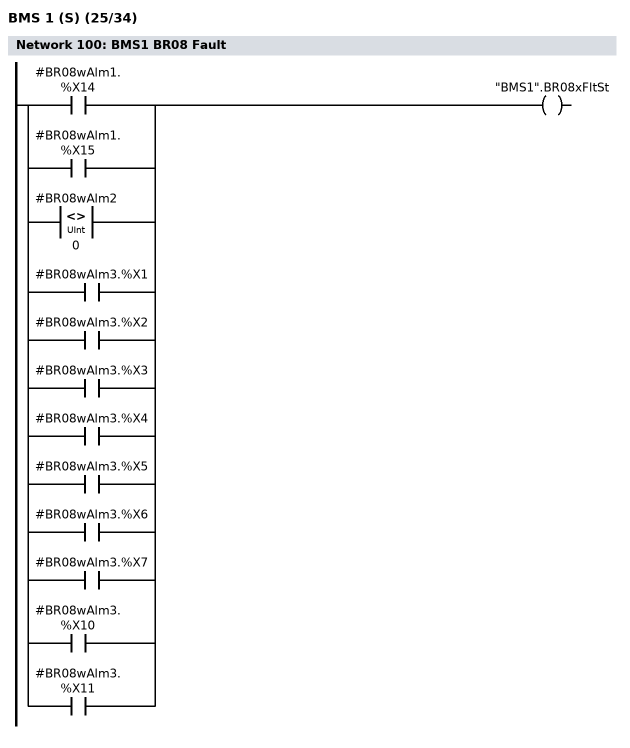
   RUNG wire#powerrail
      Contact( #BR08wAlm1.%X14 )
      wire#w1
      Coil( "BMS1".BR08xFltSt )
   END_RUNG
   RUNG wire#powerrail
      Contact( #BR08wAlm1.%X15 )
   END_RUNG wire#w1
   RUNG wire#powerrail
      { S7_Templates := "SrcType := UInt" } NE_Contact(in1 := #BR08wAlm2, in2 := 0)
   END_RUNG wire#w1
   RUNG wire#powerrail
      Contact( #BR08wAlm3.%X1 )
   END_RUNG wire#w1
   RUNG wire#powerrail
      Contact( #BR08wAlm3.%X2 )
   END_RUNG wire#w1
   RUNG wire#powerrail
      Contact( #BR08wAlm3.%X3 )
   END_RUNG wire#w1
   RUNG wire#powerrail
      Contact( #BR08wAlm3.%X4 )
   END_RUNG wire#w1
   RUNG wire#powerrail
      Contact( #BR08wAlm3.%X5 )
   END_RUNG wire#w1
   RUNG wire#powerrail
      Contact( #BR08wAlm3.%X6 )
   END_RUNG wire#w1
   RUNG wire#powerrail
      Contact( #BR08wAlm3.%X7 )
   END_RUNG wire#w1
   RUNG wire#powerrail
      Contact( #BR08wAlm3.%X10 )
   END_RUNG wire#w1
   RUNG wire#powerrail
      Contact( #BR08wAlm3.%X11 )
   END_RUNG wire#w1
   // the same network as SCL:
   "BMS1".BR08xFltSt := #BR08wAlm1.%X14 OR #BR08wAlm1.%X15 OR (#BR08wAlm2 <> 0) OR #BR08wAlm3.%X1 OR #BR08wAlm3.%X2 OR #BR08wAlm3.%X3 OR #BR08wAlm3.%X4 OR #BR08wAlm3.%X5 OR #BR08wAlm3.%X6 OR #BR08wAlm3.%X7 OR #BR08wAlm3.%X10 OR #BR08wAlm3.%X11;
END_REGION

REGION Network 101: BMS1 BR08 Alarm
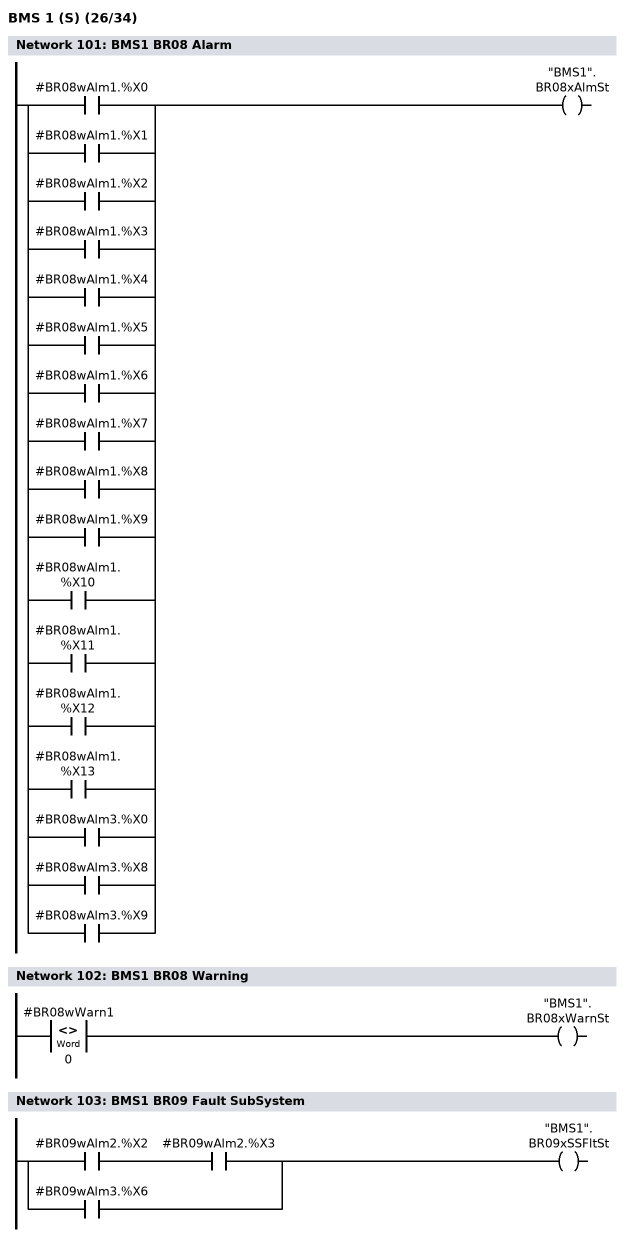
   RUNG wire#powerrail
      Contact( #BR08wAlm1.%X0 )
      wire#w1
      Coil( "BMS1".BR08xAlmSt )
   END_RUNG
   RUNG wire#powerrail
      Contact( #BR08wAlm1.%X1 )
   END_RUNG wire#w1
   RUNG wire#powerrail
      Contact( #BR08wAlm1.%X2 )
   END_RUNG wire#w1
   RUNG wire#powerrail
      Contact( #BR08wAlm1.%X3 )
   END_RUNG wire#w1
   RUNG wire#powerrail
      Contact( #BR08wAlm1.%X4 )
   END_RUNG wire#w1
   RUNG wire#powerrail
      Contact( #BR08wAlm1.%X5 )
   END_RUNG wire#w1
   RUNG wire#powerrail
      Contact( #BR08wAlm1.%X6 )
   END_RUNG wire#w1
   RUNG wire#powerrail
      Contact( #BR08wAlm1.%X7 )
   END_RUNG wire#w1
   RUNG wire#powerrail
      Contact( #BR08wAlm1.%X8 )
   END_RUNG wire#w1
   RUNG wire#powerrail
      Contact( #BR08wAlm1.%X9 )
   END_RUNG wire#w1
   RUNG wire#powerrail
      Contact( #BR08wAlm1.%X10 )
   END_RUNG wire#w1
   RUNG wire#powerrail
      Contact( #BR08wAlm1.%X11 )
   END_RUNG wire#w1
   RUNG wire#powerrail
      Contact( #BR08wAlm1.%X12 )
   END_RUNG wire#w1
   RUNG wire#powerrail
      Contact( #BR08wAlm1.%X13 )
   END_RUNG wire#w1
   RUNG wire#powerrail
      Contact( #BR08wAlm3.%X0 )
   END_RUNG wire#w1
   RUNG wire#powerrail
      Contact( #BR08wAlm3.%X8 )
   END_RUNG wire#w1
   RUNG wire#powerrail
      Contact( #BR08wAlm3.%X9 )
   END_RUNG wire#w1
   // the same network as SCL:
   "BMS1".BR08xAlmSt := #BR08wAlm1.%X0 OR #BR08wAlm1.%X1 OR #BR08wAlm1.%X2 OR #BR08wAlm1.%X3 OR #BR08wAlm1.%X4 OR #BR08wAlm1.%X5 OR #BR08wAlm1.%X6 OR #BR08wAlm1.%X7 OR #BR08wAlm1.%X8 OR #BR08wAlm1.%X9 OR #BR08wAlm1.%X10 OR #BR08wAlm1.%X11 OR #BR08wAlm1.%X12 OR #BR08wAlm1.%X13 OR #BR08wAlm3.%X0 OR #BR08wAlm3.%X8 OR #BR08wAlm3.%X9;
END_REGION

REGION Network 102: BMS1 BR08 Warning
   RUNG wire#powerrail
      { S7_Templates := "SrcType := Word" } NE_Contact(in1 := #BR08wWarn1, in2 := 0)
      Coil( "BMS1".BR08xWarnSt )
   END_RUNG
   // the same network as SCL:
   "BMS1".BR08xWarnSt := #BR08wWarn1 <> 0;
END_REGION

REGION Network 103: BMS1 BR09 Fault SubSystem
   RUNG wire#powerrail
      Contact( #BR09wAlm2.%X2 )
      Contact( #BR09wAlm2.%X3 )
      wire#w1
      Coil( "BMS1".BR09xSSFltSt )
   END_RUNG
   RUNG wire#powerrail
      Contact( #BR09wAlm3.%X6 )
   END_RUNG wire#w1
   // the same network as SCL:
   "BMS1".BR09xSSFltSt := (#BR09wAlm2.%X2 AND #BR09wAlm2.%X3) OR #BR09wAlm3.%X6;
END_REGION

REGION Network 104: BMS1 BR09 Fault
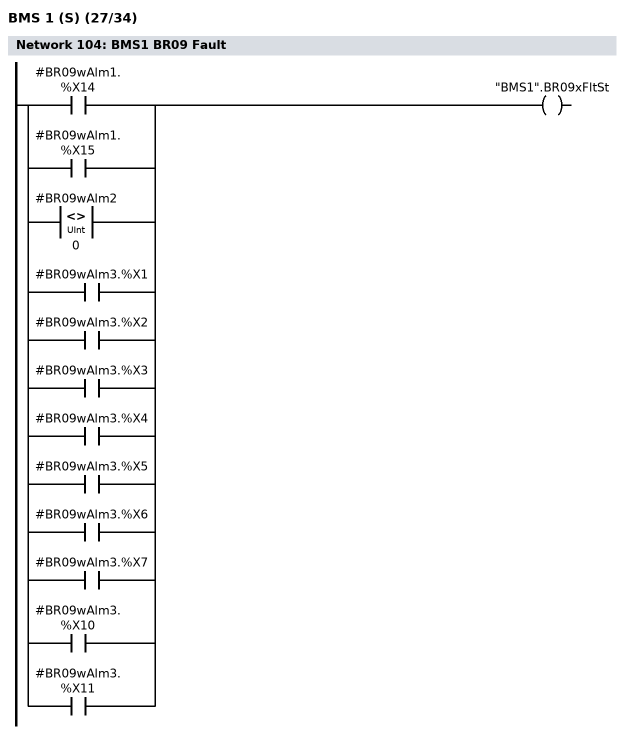
   RUNG wire#powerrail
      Contact( #BR09wAlm1.%X14 )
      wire#w1
      Coil( "BMS1".BR09xFltSt )
   END_RUNG
   RUNG wire#powerrail
      Contact( #BR09wAlm1.%X15 )
   END_RUNG wire#w1
   RUNG wire#powerrail
      { S7_Templates := "SrcType := UInt" } NE_Contact(in1 := #BR09wAlm2, in2 := 0)
   END_RUNG wire#w1
   RUNG wire#powerrail
      Contact( #BR09wAlm3.%X1 )
   END_RUNG wire#w1
   RUNG wire#powerrail
      Contact( #BR09wAlm3.%X2 )
   END_RUNG wire#w1
   RUNG wire#powerrail
      Contact( #BR09wAlm3.%X3 )
   END_RUNG wire#w1
   RUNG wire#powerrail
      Contact( #BR09wAlm3.%X4 )
   END_RUNG wire#w1
   RUNG wire#powerrail
      Contact( #BR09wAlm3.%X5 )
   END_RUNG wire#w1
   RUNG wire#powerrail
      Contact( #BR09wAlm3.%X6 )
   END_RUNG wire#w1
   RUNG wire#powerrail
      Contact( #BR09wAlm3.%X7 )
   END_RUNG wire#w1
   RUNG wire#powerrail
      Contact( #BR09wAlm3.%X10 )
   END_RUNG wire#w1
   RUNG wire#powerrail
      Contact( #BR09wAlm3.%X11 )
   END_RUNG wire#w1
   // the same network as SCL:
   "BMS1".BR09xFltSt := #BR09wAlm1.%X14 OR #BR09wAlm1.%X15 OR (#BR09wAlm2 <> 0) OR #BR09wAlm3.%X1 OR #BR09wAlm3.%X2 OR #BR09wAlm3.%X3 OR #BR09wAlm3.%X4 OR #BR09wAlm3.%X5 OR #BR09wAlm3.%X6 OR #BR09wAlm3.%X7 OR #BR09wAlm3.%X10 OR #BR09wAlm3.%X11;
END_REGION

REGION Network 105: BMS1 BR09 Alarm
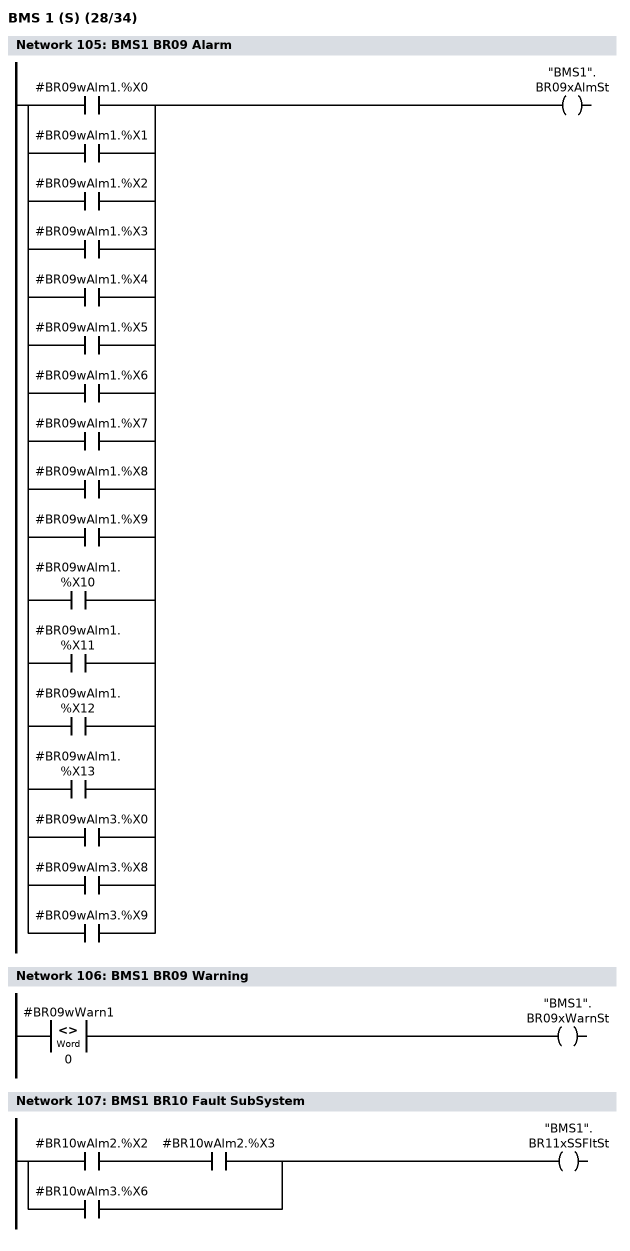
   RUNG wire#powerrail
      Contact( #BR09wAlm1.%X0 )
      wire#w1
      Coil( "BMS1".BR09xAlmSt )
   END_RUNG
   RUNG wire#powerrail
      Contact( #BR09wAlm1.%X1 )
   END_RUNG wire#w1
   RUNG wire#powerrail
      Contact( #BR09wAlm1.%X2 )
   END_RUNG wire#w1
   RUNG wire#powerrail
      Contact( #BR09wAlm1.%X3 )
   END_RUNG wire#w1
   RUNG wire#powerrail
      Contact( #BR09wAlm1.%X4 )
   END_RUNG wire#w1
   RUNG wire#powerrail
      Contact( #BR09wAlm1.%X5 )
   END_RUNG wire#w1
   RUNG wire#powerrail
      Contact( #BR09wAlm1.%X6 )
   END_RUNG wire#w1
   RUNG wire#powerrail
      Contact( #BR09wAlm1.%X7 )
   END_RUNG wire#w1
   RUNG wire#powerrail
      Contact( #BR09wAlm1.%X8 )
   END_RUNG wire#w1
   RUNG wire#powerrail
      Contact( #BR09wAlm1.%X9 )
   END_RUNG wire#w1
   RUNG wire#powerrail
      Contact( #BR09wAlm1.%X10 )
   END_RUNG wire#w1
   RUNG wire#powerrail
      Contact( #BR09wAlm1.%X11 )
   END_RUNG wire#w1
   RUNG wire#powerrail
      Contact( #BR09wAlm1.%X12 )
   END_RUNG wire#w1
   RUNG wire#powerrail
      Contact( #BR09wAlm1.%X13 )
   END_RUNG wire#w1
   RUNG wire#powerrail
      Contact( #BR09wAlm3.%X0 )
   END_RUNG wire#w1
   RUNG wire#powerrail
      Contact( #BR09wAlm3.%X8 )
   END_RUNG wire#w1
   RUNG wire#powerrail
      Contact( #BR09wAlm3.%X9 )
   END_RUNG wire#w1
   // the same network as SCL:
   "BMS1".BR09xAlmSt := #BR09wAlm1.%X0 OR #BR09wAlm1.%X1 OR #BR09wAlm1.%X2 OR #BR09wAlm1.%X3 OR #BR09wAlm1.%X4 OR #BR09wAlm1.%X5 OR #BR09wAlm1.%X6 OR #BR09wAlm1.%X7 OR #BR09wAlm1.%X8 OR #BR09wAlm1.%X9 OR #BR09wAlm1.%X10 OR #BR09wAlm1.%X11 OR #BR09wAlm1.%X12 OR #BR09wAlm1.%X13 OR #BR09wAlm3.%X0 OR #BR09wAlm3.%X8 OR #BR09wAlm3.%X9;
END_REGION

REGION Network 106: BMS1 BR09 Warning
   RUNG wire#powerrail
      { S7_Templates := "SrcType := Word" } NE_Contact(in1 := #BR09wWarn1, in2 := 0)
      Coil( "BMS1".BR09xWarnSt )
   END_RUNG
   // the same network as SCL:
   "BMS1".BR09xWarnSt := #BR09wWarn1 <> 0;
END_REGION

REGION Network 107: BMS1 BR10 Fault SubSystem
   RUNG wire#powerrail
      Contact( #BR10wAlm2.%X2 )
      Contact( #BR10wAlm2.%X3 )
      wire#w1
      Coil( "BMS1".BR11xSSFltSt )
   END_RUNG
   RUNG wire#powerrail
      Contact( #BR10wAlm3.%X6 )
   END_RUNG wire#w1
   // the same network as SCL:
   "BMS1".BR11xSSFltSt := (#BR10wAlm2.%X2 AND #BR10wAlm2.%X3) OR #BR10wAlm3.%X6;
END_REGION

REGION Network 108: BMS1 BR10 Fault
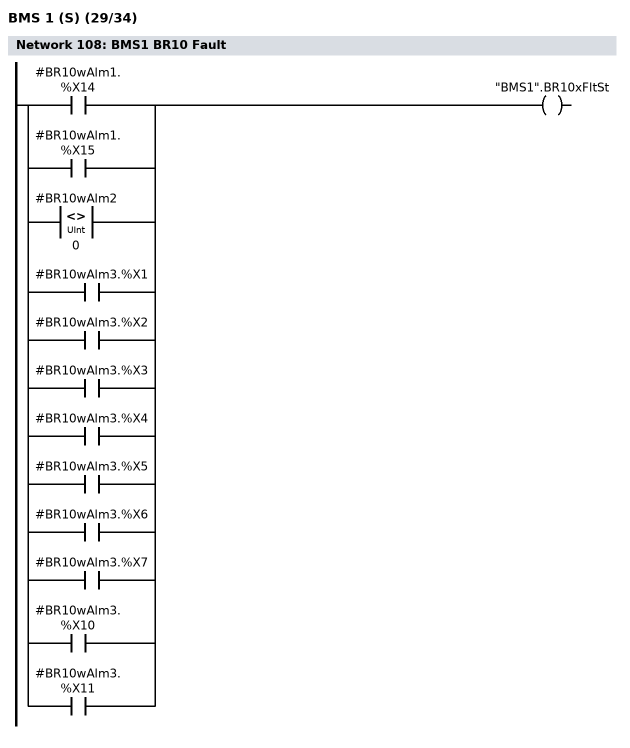
   RUNG wire#powerrail
      Contact( #BR10wAlm1.%X14 )
      wire#w1
      Coil( "BMS1".BR10xFltSt )
   END_RUNG
   RUNG wire#powerrail
      Contact( #BR10wAlm1.%X15 )
   END_RUNG wire#w1
   RUNG wire#powerrail
      { S7_Templates := "SrcType := UInt" } NE_Contact(in1 := #BR10wAlm2, in2 := 0)
   END_RUNG wire#w1
   RUNG wire#powerrail
      Contact( #BR10wAlm3.%X1 )
   END_RUNG wire#w1
   RUNG wire#powerrail
      Contact( #BR10wAlm3.%X2 )
   END_RUNG wire#w1
   RUNG wire#powerrail
      Contact( #BR10wAlm3.%X3 )
   END_RUNG wire#w1
   RUNG wire#powerrail
      Contact( #BR10wAlm3.%X4 )
   END_RUNG wire#w1
   RUNG wire#powerrail
      Contact( #BR10wAlm3.%X5 )
   END_RUNG wire#w1
   RUNG wire#powerrail
      Contact( #BR10wAlm3.%X6 )
   END_RUNG wire#w1
   RUNG wire#powerrail
      Contact( #BR10wAlm3.%X7 )
   END_RUNG wire#w1
   RUNG wire#powerrail
      Contact( #BR10wAlm3.%X10 )
   END_RUNG wire#w1
   RUNG wire#powerrail
      Contact( #BR10wAlm3.%X11 )
   END_RUNG wire#w1
   // the same network as SCL:
   "BMS1".BR10xFltSt := #BR10wAlm1.%X14 OR #BR10wAlm1.%X15 OR (#BR10wAlm2 <> 0) OR #BR10wAlm3.%X1 OR #BR10wAlm3.%X2 OR #BR10wAlm3.%X3 OR #BR10wAlm3.%X4 OR #BR10wAlm3.%X5 OR #BR10wAlm3.%X6 OR #BR10wAlm3.%X7 OR #BR10wAlm3.%X10 OR #BR10wAlm3.%X11;
END_REGION

REGION Network 109: BMS1 BR10 Alarm
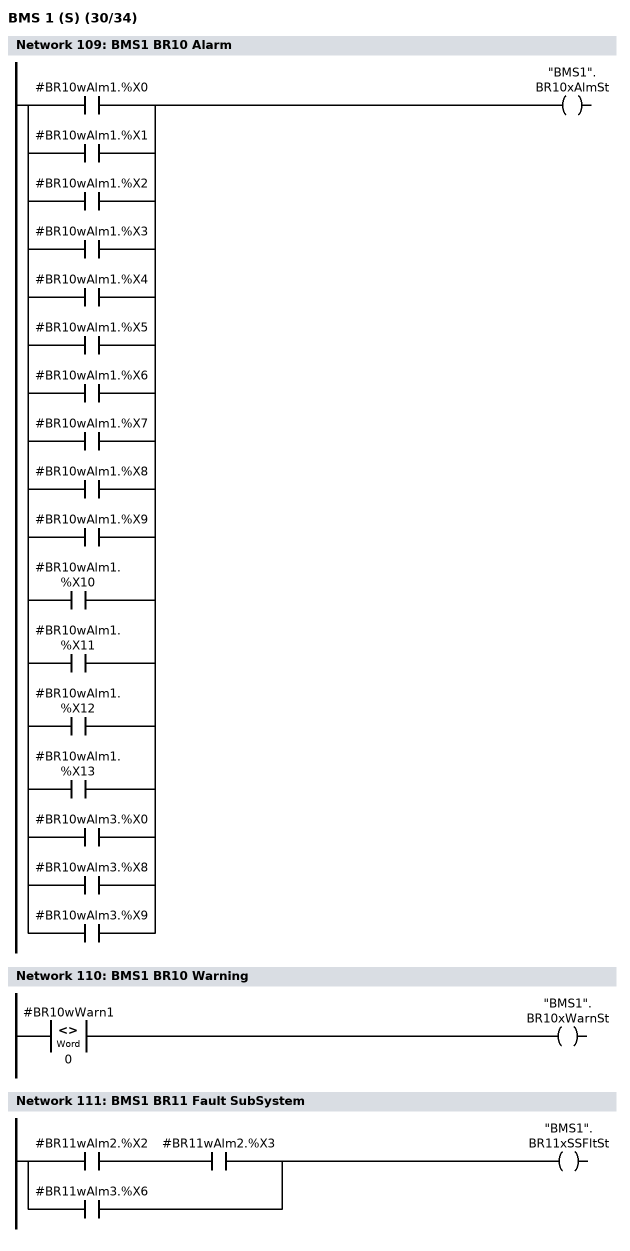
   RUNG wire#powerrail
      Contact( #BR10wAlm1.%X0 )
      wire#w1
      Coil( "BMS1".BR10xAlmSt )
   END_RUNG
   RUNG wire#powerrail
      Contact( #BR10wAlm1.%X1 )
   END_RUNG wire#w1
   RUNG wire#powerrail
      Contact( #BR10wAlm1.%X2 )
   END_RUNG wire#w1
   RUNG wire#powerrail
      Contact( #BR10wAlm1.%X3 )
   END_RUNG wire#w1
   RUNG wire#powerrail
      Contact( #BR10wAlm1.%X4 )
   END_RUNG wire#w1
   RUNG wire#powerrail
      Contact( #BR10wAlm1.%X5 )
   END_RUNG wire#w1
   RUNG wire#powerrail
      Contact( #BR10wAlm1.%X6 )
   END_RUNG wire#w1
   RUNG wire#powerrail
      Contact( #BR10wAlm1.%X7 )
   END_RUNG wire#w1
   RUNG wire#powerrail
      Contact( #BR10wAlm1.%X8 )
   END_RUNG wire#w1
   RUNG wire#powerrail
      Contact( #BR10wAlm1.%X9 )
   END_RUNG wire#w1
   RUNG wire#powerrail
      Contact( #BR10wAlm1.%X10 )
   END_RUNG wire#w1
   RUNG wire#powerrail
      Contact( #BR10wAlm1.%X11 )
   END_RUNG wire#w1
   RUNG wire#powerrail
      Contact( #BR10wAlm1.%X12 )
   END_RUNG wire#w1
   RUNG wire#powerrail
      Contact( #BR10wAlm1.%X13 )
   END_RUNG wire#w1
   RUNG wire#powerrail
      Contact( #BR10wAlm3.%X0 )
   END_RUNG wire#w1
   RUNG wire#powerrail
      Contact( #BR10wAlm3.%X8 )
   END_RUNG wire#w1
   RUNG wire#powerrail
      Contact( #BR10wAlm3.%X9 )
   END_RUNG wire#w1
   // the same network as SCL:
   "BMS1".BR10xAlmSt := #BR10wAlm1.%X0 OR #BR10wAlm1.%X1 OR #BR10wAlm1.%X2 OR #BR10wAlm1.%X3 OR #BR10wAlm1.%X4 OR #BR10wAlm1.%X5 OR #BR10wAlm1.%X6 OR #BR10wAlm1.%X7 OR #BR10wAlm1.%X8 OR #BR10wAlm1.%X9 OR #BR10wAlm1.%X10 OR #BR10wAlm1.%X11 OR #BR10wAlm1.%X12 OR #BR10wAlm1.%X13 OR #BR10wAlm3.%X0 OR #BR10wAlm3.%X8 OR #BR10wAlm3.%X9;
END_REGION

REGION Network 110: BMS1 BR10 Warning
   RUNG wire#powerrail
      { S7_Templates := "SrcType := Word" } NE_Contact(in1 := #BR10wWarn1, in2 := 0)
      Coil( "BMS1".BR10xWarnSt )
   END_RUNG
   // the same network as SCL:
   "BMS1".BR10xWarnSt := #BR10wWarn1 <> 0;
END_REGION

REGION Network 111: BMS1 BR11 Fault SubSystem
   RUNG wire#powerrail
      Contact( #BR11wAlm2.%X2 )
      Contact( #BR11wAlm2.%X3 )
      wire#w1
      Coil( "BMS1".BR11xSSFltSt )
   END_RUNG
   RUNG wire#powerrail
      Contact( #BR11wAlm3.%X6 )
   END_RUNG wire#w1
   // the same network as SCL:
   "BMS1".BR11xSSFltSt := (#BR11wAlm2.%X2 AND #BR11wAlm2.%X3) OR #BR11wAlm3.%X6;
END_REGION

REGION Network 112: BMS1 BR11 Fault
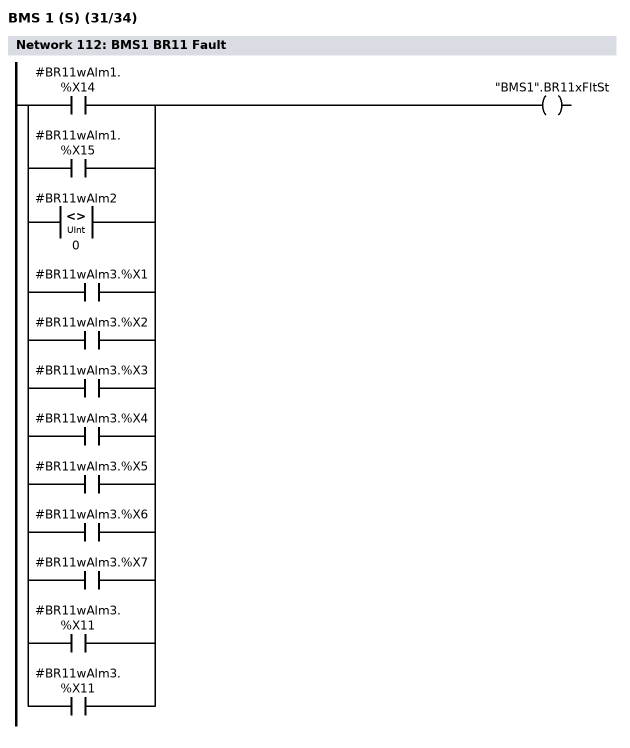
   RUNG wire#powerrail
      Contact( #BR11wAlm1.%X14 )
      wire#w1
      Coil( "BMS1".BR11xFltSt )
   END_RUNG
   RUNG wire#powerrail
      Contact( #BR11wAlm1.%X15 )
   END_RUNG wire#w1
   RUNG wire#powerrail
      { S7_Templates := "SrcType := UInt" } NE_Contact(in1 := #BR11wAlm2, in2 := 0)
   END_RUNG wire#w1
   RUNG wire#powerrail
      Contact( #BR11wAlm3.%X1 )
   END_RUNG wire#w1
   RUNG wire#powerrail
      Contact( #BR11wAlm3.%X2 )
   END_RUNG wire#w1
   RUNG wire#powerrail
      Contact( #BR11wAlm3.%X3 )
   END_RUNG wire#w1
   RUNG wire#powerrail
      Contact( #BR11wAlm3.%X4 )
   END_RUNG wire#w1
   RUNG wire#powerrail
      Contact( #BR11wAlm3.%X5 )
   END_RUNG wire#w1
   RUNG wire#powerrail
      Contact( #BR11wAlm3.%X6 )
   END_RUNG wire#w1
   RUNG wire#powerrail
      Contact( #BR11wAlm3.%X7 )
   END_RUNG wire#w1
   RUNG wire#powerrail
      Contact( #BR11wAlm3.%X11 )
   END_RUNG wire#w1
   RUNG wire#powerrail
      Contact( #BR11wAlm3.%X11 )
   END_RUNG wire#w1
   // the same network as SCL:
   "BMS1".BR11xFltSt := #BR11wAlm1.%X14 OR #BR11wAlm1.%X15 OR (#BR11wAlm2 <> 0) OR #BR11wAlm3.%X1 OR #BR11wAlm3.%X2 OR #BR11wAlm3.%X3 OR #BR11wAlm3.%X4 OR #BR11wAlm3.%X5 OR #BR11wAlm3.%X6 OR #BR11wAlm3.%X7 OR #BR11wAlm3.%X11 OR #BR11wAlm3.%X11;
END_REGION

REGION Network 113: BMS1 BR11 Alarm
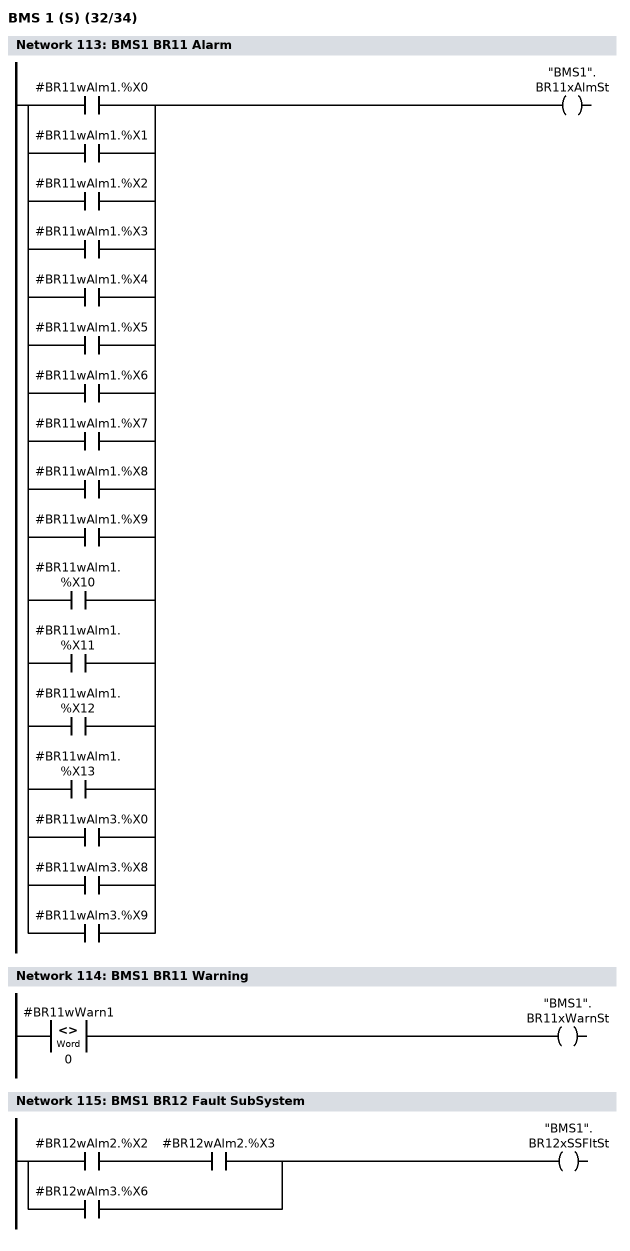
   RUNG wire#powerrail
      Contact( #BR11wAlm1.%X0 )
      wire#w1
      Coil( "BMS1".BR11xAlmSt )
   END_RUNG
   RUNG wire#powerrail
      Contact( #BR11wAlm1.%X1 )
   END_RUNG wire#w1
   RUNG wire#powerrail
      Contact( #BR11wAlm1.%X2 )
   END_RUNG wire#w1
   RUNG wire#powerrail
      Contact( #BR11wAlm1.%X3 )
   END_RUNG wire#w1
   RUNG wire#powerrail
      Contact( #BR11wAlm1.%X4 )
   END_RUNG wire#w1
   RUNG wire#powerrail
      Contact( #BR11wAlm1.%X5 )
   END_RUNG wire#w1
   RUNG wire#powerrail
      Contact( #BR11wAlm1.%X6 )
   END_RUNG wire#w1
   RUNG wire#powerrail
      Contact( #BR11wAlm1.%X7 )
   END_RUNG wire#w1
   RUNG wire#powerrail
      Contact( #BR11wAlm1.%X8 )
   END_RUNG wire#w1
   RUNG wire#powerrail
      Contact( #BR11wAlm1.%X9 )
   END_RUNG wire#w1
   RUNG wire#powerrail
      Contact( #BR11wAlm1.%X10 )
   END_RUNG wire#w1
   RUNG wire#powerrail
      Contact( #BR11wAlm1.%X11 )
   END_RUNG wire#w1
   RUNG wire#powerrail
      Contact( #BR11wAlm1.%X12 )
   END_RUNG wire#w1
   RUNG wire#powerrail
      Contact( #BR11wAlm1.%X13 )
   END_RUNG wire#w1
   RUNG wire#powerrail
      Contact( #BR11wAlm3.%X0 )
   END_RUNG wire#w1
   RUNG wire#powerrail
      Contact( #BR11wAlm3.%X8 )
   END_RUNG wire#w1
   RUNG wire#powerrail
      Contact( #BR11wAlm3.%X9 )
   END_RUNG wire#w1
   // the same network as SCL:
   "BMS1".BR11xAlmSt := #BR11wAlm1.%X0 OR #BR11wAlm1.%X1 OR #BR11wAlm1.%X2 OR #BR11wAlm1.%X3 OR #BR11wAlm1.%X4 OR #BR11wAlm1.%X5 OR #BR11wAlm1.%X6 OR #BR11wAlm1.%X7 OR #BR11wAlm1.%X8 OR #BR11wAlm1.%X9 OR #BR11wAlm1.%X10 OR #BR11wAlm1.%X11 OR #BR11wAlm1.%X12 OR #BR11wAlm1.%X13 OR #BR11wAlm3.%X0 OR #BR11wAlm3.%X8 OR #BR11wAlm3.%X9;
END_REGION

REGION Network 114: BMS1 BR11 Warning
   RUNG wire#powerrail
      { S7_Templates := "SrcType := Word" } NE_Contact(in1 := #BR11wWarn1, in2 := 0)
      Coil( "BMS1".BR11xWarnSt )
   END_RUNG
   // the same network as SCL:
   "BMS1".BR11xWarnSt := #BR11wWarn1 <> 0;
END_REGION

REGION Network 115: BMS1 BR12 Fault SubSystem
   RUNG wire#powerrail
      Contact( #BR12wAlm2.%X2 )
      Contact( #BR12wAlm2.%X3 )
      wire#w1
      Coil( "BMS1".BR12xSSFltSt )
   END_RUNG
   RUNG wire#powerrail
      Contact( #BR12wAlm3.%X6 )
   END_RUNG wire#w1
   // the same network as SCL:
   "BMS1".BR12xSSFltSt := (#BR12wAlm2.%X2 AND #BR12wAlm2.%X3) OR #BR12wAlm3.%X6;
END_REGION

REGION Network 116: BMS1 BR12 Fault
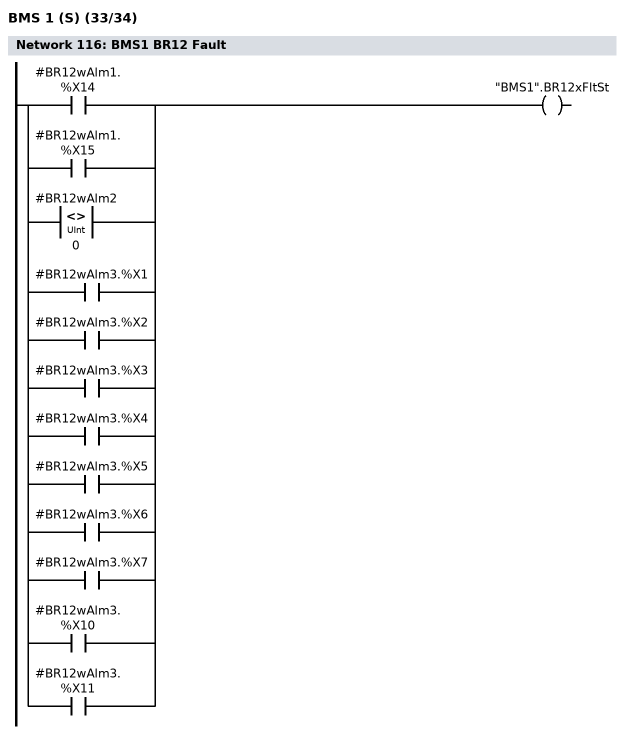
   RUNG wire#powerrail
      Contact( #BR12wAlm1.%X14 )
      wire#w1
      Coil( "BMS1".BR12xFltSt )
   END_RUNG
   RUNG wire#powerrail
      Contact( #BR12wAlm1.%X15 )
   END_RUNG wire#w1
   RUNG wire#powerrail
      { S7_Templates := "SrcType := UInt" } NE_Contact(in1 := #BR12wAlm2, in2 := 0)
   END_RUNG wire#w1
   RUNG wire#powerrail
      Contact( #BR12wAlm3.%X1 )
   END_RUNG wire#w1
   RUNG wire#powerrail
      Contact( #BR12wAlm3.%X2 )
   END_RUNG wire#w1
   RUNG wire#powerrail
      Contact( #BR12wAlm3.%X3 )
   END_RUNG wire#w1
   RUNG wire#powerrail
      Contact( #BR12wAlm3.%X4 )
   END_RUNG wire#w1
   RUNG wire#powerrail
      Contact( #BR12wAlm3.%X5 )
   END_RUNG wire#w1
   RUNG wire#powerrail
      Contact( #BR12wAlm3.%X6 )
   END_RUNG wire#w1
   RUNG wire#powerrail
      Contact( #BR12wAlm3.%X7 )
   END_RUNG wire#w1
   RUNG wire#powerrail
      Contact( #BR12wAlm3.%X10 )
   END_RUNG wire#w1
   RUNG wire#powerrail
      Contact( #BR12wAlm3.%X11 )
   END_RUNG wire#w1
   // the same network as SCL:
   "BMS1".BR12xFltSt := #BR12wAlm1.%X14 OR #BR12wAlm1.%X15 OR (#BR12wAlm2 <> 0) OR #BR12wAlm3.%X1 OR #BR12wAlm3.%X2 OR #BR12wAlm3.%X3 OR #BR12wAlm3.%X4 OR #BR12wAlm3.%X5 OR #BR12wAlm3.%X6 OR #BR12wAlm3.%X7 OR #BR12wAlm3.%X10 OR #BR12wAlm3.%X11;
END_REGION

REGION Network 117: BMS1 BR12 Alarm
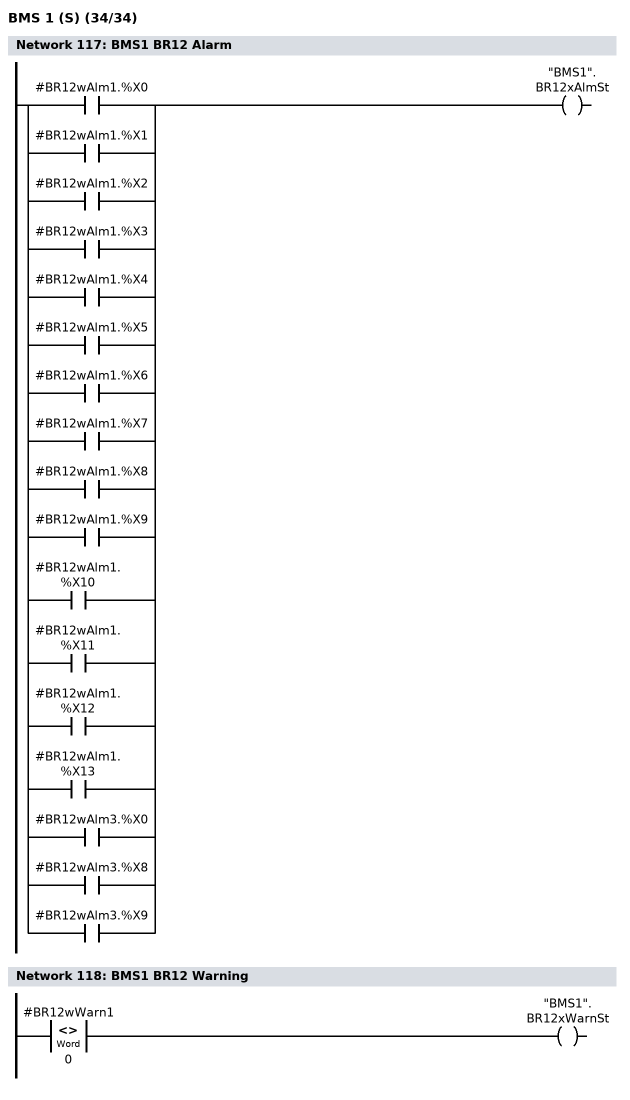
   RUNG wire#powerrail
      Contact( #BR12wAlm1.%X0 )
      wire#w1
      Coil( "BMS1".BR12xAlmSt )
   END_RUNG
   RUNG wire#powerrail
      Contact( #BR12wAlm1.%X1 )
   END_RUNG wire#w1
   RUNG wire#powerrail
      Contact( #BR12wAlm1.%X2 )
   END_RUNG wire#w1
   RUNG wire#powerrail
      Contact( #BR12wAlm1.%X3 )
   END_RUNG wire#w1
   RUNG wire#powerrail
      Contact( #BR12wAlm1.%X4 )
   END_RUNG wire#w1
   RUNG wire#powerrail
      Contact( #BR12wAlm1.%X5 )
   END_RUNG wire#w1
   RUNG wire#powerrail
      Contact( #BR12wAlm1.%X6 )
   END_RUNG wire#w1
   RUNG wire#powerrail
      Contact( #BR12wAlm1.%X7 )
   END_RUNG wire#w1
   RUNG wire#powerrail
      Contact( #BR12wAlm1.%X8 )
   END_RUNG wire#w1
   RUNG wire#powerrail
      Contact( #BR12wAlm1.%X9 )
   END_RUNG wire#w1
   RUNG wire#powerrail
      Contact( #BR12wAlm1.%X10 )
   END_RUNG wire#w1
   RUNG wire#powerrail
      Contact( #BR12wAlm1.%X11 )
   END_RUNG wire#w1
   RUNG wire#powerrail
      Contact( #BR12wAlm1.%X12 )
   END_RUNG wire#w1
   RUNG wire#powerrail
      Contact( #BR12wAlm1.%X13 )
   END_RUNG wire#w1
   RUNG wire#powerrail
      Contact( #BR12wAlm3.%X0 )
   END_RUNG wire#w1
   RUNG wire#powerrail
      Contact( #BR12wAlm3.%X8 )
   END_RUNG wire#w1
   RUNG wire#powerrail
      Contact( #BR12wAlm3.%X9 )
   END_RUNG wire#w1
   // the same network as SCL:
   "BMS1".BR12xAlmSt := #BR12wAlm1.%X0 OR #BR12wAlm1.%X1 OR #BR12wAlm1.%X2 OR #BR12wAlm1.%X3 OR #BR12wAlm1.%X4 OR #BR12wAlm1.%X5 OR #BR12wAlm1.%X6 OR #BR12wAlm1.%X7 OR #BR12wAlm1.%X8 OR #BR12wAlm1.%X9 OR #BR12wAlm1.%X10 OR #BR12wAlm1.%X11 OR #BR12wAlm1.%X12 OR #BR12wAlm1.%X13 OR #BR12wAlm3.%X0 OR #BR12wAlm3.%X8 OR #BR12wAlm3.%X9;
END_REGION

REGION Network 118: BMS1 BR12 Warning
   RUNG wire#powerrail
      { S7_Templates := "SrcType := Word" } NE_Contact(in1 := #BR12wWarn1, in2 := 0)
      Coil( "BMS1".BR12xWarnSt )
   END_RUNG
   // the same network as SCL:
   "BMS1".BR12xWarnSt := #BR12wWarn1 <> 0;
END_REGION
END_FUNCTION
